FUNCTION_BLOCK FB_SecondOrderHold
VAR_INPUT
	u_k		: REAL; // Eingangswert
	T		: REAL;	// Zeitkonstante
	d		: REAL; // Daempfung
	w0		: REAL; // Eigenfrequenz 
END_VAR
VAR_OUTPUT
	y_k		: REAL; // Ausgangswert
END_VAR
VAR
	a		: REAL; // Variable fuer w0^2 * T^2
	b 		: REAL; // Variable fuer 2 * d * w0 * T
	y_k_1	: REAL; // letzer Ausgangswert
	y_k_2	: REAL; // vorletzer Ausgangswert
END_VAR

a := (w0 * w0) * (T * T);
b := 2 * d * w0 * T; 

y_k := (u_k*a + 2*y_k_1 + b*y_k_1 - y_k_2) / (1 + b + a); 

y_k_2 := y_k_1;
y_k_1 := y_k;

END_FUNCTION_BLOCK

(* stored: Version 1.1.0.1, ProductVersion 3.1.4024.9
   POU FB_SecondOrderHold: Id {7226bd99-01fe-4b1d-bd86-8d10e11cde16}, SpecialFunc None *)
